FUNCTION_BLOCK FB_SplitFloatToWords
////////////////// 
// Merge two words into a real with IEEE 754 coding (for float reading). 
//////////////////	
VAR_INPUT
	
	VAR_IN 		AT %MD0 : REAL;
END_VAR

VAR_OUTPUT
	
	WORD_STRONG 	AT %MW1 : WORD; // Strong Word 
	WORD_WEAK 	AT %MW0 : WORD; // Weak Word. 
END_VAR

END_FUNCTION_BLOCK

(* stored: Version 1.1.0.1, ProductVersion 3.1.4024.6
   POU FB_SplitFloatToWords: Id {0e90db96-f810-4b27-9644-c6409196c32a}, SpecialFunc None *)
